Fanuc KAREL source: ka00068.KL

PROGRAM KA00068
%STACKSIZE=65535
%PRIORITY=65535
%NOLOCKGROUP
VAR
SRC : XYZWPR
DST : JOINTPOS9
BEGIN
SRC.X=1.0
-- UNSAFE_SOURCE_IR line 8: DST = convert_xyzwpr_to_jointpos9(SRC)
END KA00068
